// TIA Portal V21 export
VAR_GLOBAL   // PLC tag table "InputAnalogici"
END_VAR
